// TIA Portal V18 export
FUNCTION_BLOCK "ST10_StopperCtrl"   // FB2601, LAD
TITLE = 输送带控制
{ S7_Optimized_Access := 'FALSE' }
VERSION : 0.1
// stored: AutoNumber false, IsIECCheckEnabled false, SetENOAutomatically false, UDAEnableTagReadback false
   VAR
      Stopper { S7_SetPoint := 'True'} : Array[1..100] of "StopperCtrl";
   END_VAR
   VAR_TEMP   // added for the SCL form of the ladder/FBD networks
      _w1 : Bool;
   END_VAR
BEGIN

REGION Network 1: ------------------------------------------------------------------------------------------------------------------------------ / ------------------------------------------------ H -------------------------------------------------------------------------
END_REGION

REGION Network 2: H-shaftLoadingStopperCylinder1
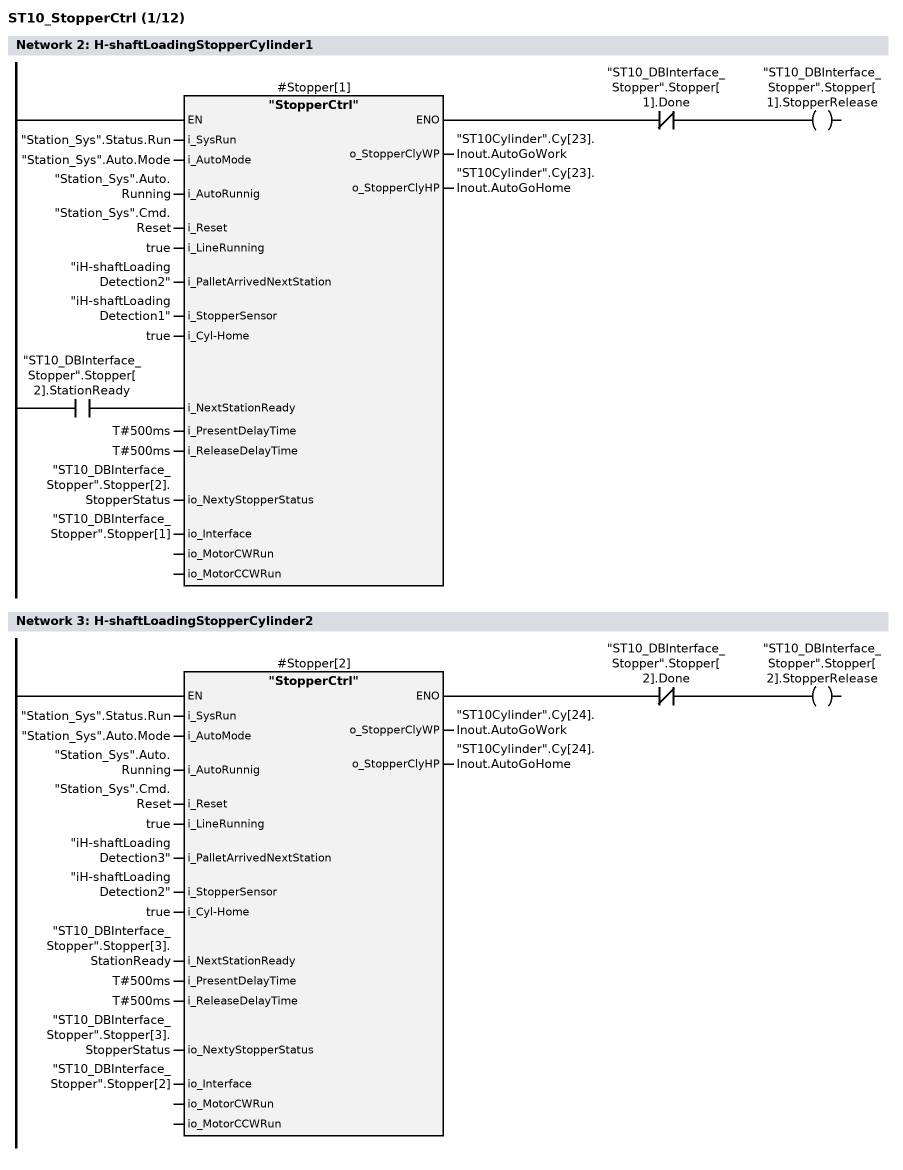
   RUNG wire#powerrail
      #Stopper[1](i_NextStationReady := wire#w1, i_SysRun := "Station_Sys".Status.Run, i_AutoMode := "Station_Sys".Auto.Mode, i_AutoRunnig := "Station_Sys".Auto.Running, i_Reset := "Station_Sys".Cmd.Reset, i_LineRunning := true, i_PalletArrivedNextStation := "iH-shaftLoadingDetection2", i_StopperSensor := "iH-shaftLoadingDetection1", "i_Cyl-Home" := true, i_PresentDelayTime := T#500ms, i_ReleaseDelayTime := T#500ms, io_NextyStopperStatus := "ST10_DBInterface_Stopper".Stopper[2].StopperStatus, io_Interface := "ST10_DBInterface_Stopper".Stopper[1], io_MotorCWRun :=, io_MotorCCWRun :=, o_StopperClyWP => "ST10Cylinder".Cy[23].Inout.AutoGoWork, o_StopperClyHP => "ST10Cylinder".Cy[23].Inout.AutoGoHome)
      I_Contact( "ST10_DBInterface_Stopper".Stopper[1].Done )
      Coil( "ST10_DBInterface_Stopper".Stopper[1].StopperRelease )
   END_RUNG
   RUNG wire#powerrail
      Contact( "ST10_DBInterface_Stopper".Stopper[2].StationReady )
   END_RUNG wire#w1
   // the same network as SCL:
   #Stopper[1](i_SysRun := "Station_Sys".Status.Run,   // "StopperCtrl"
               i_AutoMode := "Station_Sys".Auto.Mode,
               i_AutoRunnig := "Station_Sys".Auto.Running,
               i_Reset := "Station_Sys".Cmd.Reset,
               i_LineRunning := true,
               i_PalletArrivedNextStation := "iH-shaftLoadingDetection2",
               i_StopperSensor := "iH-shaftLoadingDetection1",
               "i_Cyl-Home" := true,
               i_NextStationReady := "ST10_DBInterface_Stopper".Stopper[2].StationReady,
               i_PresentDelayTime := T#500ms,
               i_ReleaseDelayTime := T#500ms,
               io_NextyStopperStatus := "ST10_DBInterface_Stopper".Stopper[2].StopperStatus,
               io_Interface := "ST10_DBInterface_Stopper".Stopper[1],
               o_StopperClyWP => "ST10Cylinder".Cy[23].Inout.AutoGoWork,
               o_StopperClyHP => "ST10Cylinder".Cy[23].Inout.AutoGoHome,
               ENO => #_w1);
   "ST10_DBInterface_Stopper".Stopper[1].StopperRelease := #_w1 AND NOT "ST10_DBInterface_Stopper".Stopper[1].Done;
END_REGION

REGION Network 3: H-shaftLoadingStopperCylinder2
   RUNG wire#powerrail
      #Stopper[2](i_SysRun := "Station_Sys".Status.Run, i_AutoMode := "Station_Sys".Auto.Mode, i_AutoRunnig := "Station_Sys".Auto.Running, i_Reset := "Station_Sys".Cmd.Reset, i_LineRunning := true, i_PalletArrivedNextStation := "iH-shaftLoadingDetection3", i_StopperSensor := "iH-shaftLoadingDetection2", "i_Cyl-Home" := true, i_NextStationReady := "ST10_DBInterface_Stopper".Stopper[3].StationReady, i_PresentDelayTime := T#500ms, i_ReleaseDelayTime := T#500ms, io_NextyStopperStatus := "ST10_DBInterface_Stopper".Stopper[3].StopperStatus, io_Interface := "ST10_DBInterface_Stopper".Stopper[2], io_MotorCWRun :=, io_MotorCCWRun :=, o_StopperClyWP => "ST10Cylinder".Cy[24].Inout.AutoGoWork, o_StopperClyHP => "ST10Cylinder".Cy[24].Inout.AutoGoHome)
      I_Contact( "ST10_DBInterface_Stopper".Stopper[2].Done )
      Coil( "ST10_DBInterface_Stopper".Stopper[2].StopperRelease )
   END_RUNG
   // the same network as SCL:
   #Stopper[2](i_SysRun := "Station_Sys".Status.Run,   // "StopperCtrl"
               i_AutoMode := "Station_Sys".Auto.Mode,
               i_AutoRunnig := "Station_Sys".Auto.Running,
               i_Reset := "Station_Sys".Cmd.Reset,
               i_LineRunning := true,
               i_PalletArrivedNextStation := "iH-shaftLoadingDetection3",
               i_StopperSensor := "iH-shaftLoadingDetection2",
               "i_Cyl-Home" := true,
               i_NextStationReady := "ST10_DBInterface_Stopper".Stopper[3].StationReady,
               i_PresentDelayTime := T#500ms,
               i_ReleaseDelayTime := T#500ms,
               io_NextyStopperStatus := "ST10_DBInterface_Stopper".Stopper[3].StopperStatus,
               io_Interface := "ST10_DBInterface_Stopper".Stopper[2],
               o_StopperClyWP => "ST10Cylinder".Cy[24].Inout.AutoGoWork,
               o_StopperClyHP => "ST10Cylinder".Cy[24].Inout.AutoGoHome,
               ENO => #_w1);
   "ST10_DBInterface_Stopper".Stopper[2].StopperRelease := #_w1 AND NOT "ST10_DBInterface_Stopper".Stopper[2].Done;
END_REGION

REGION Network 4: H-shaftLoadingStopperCylinder3
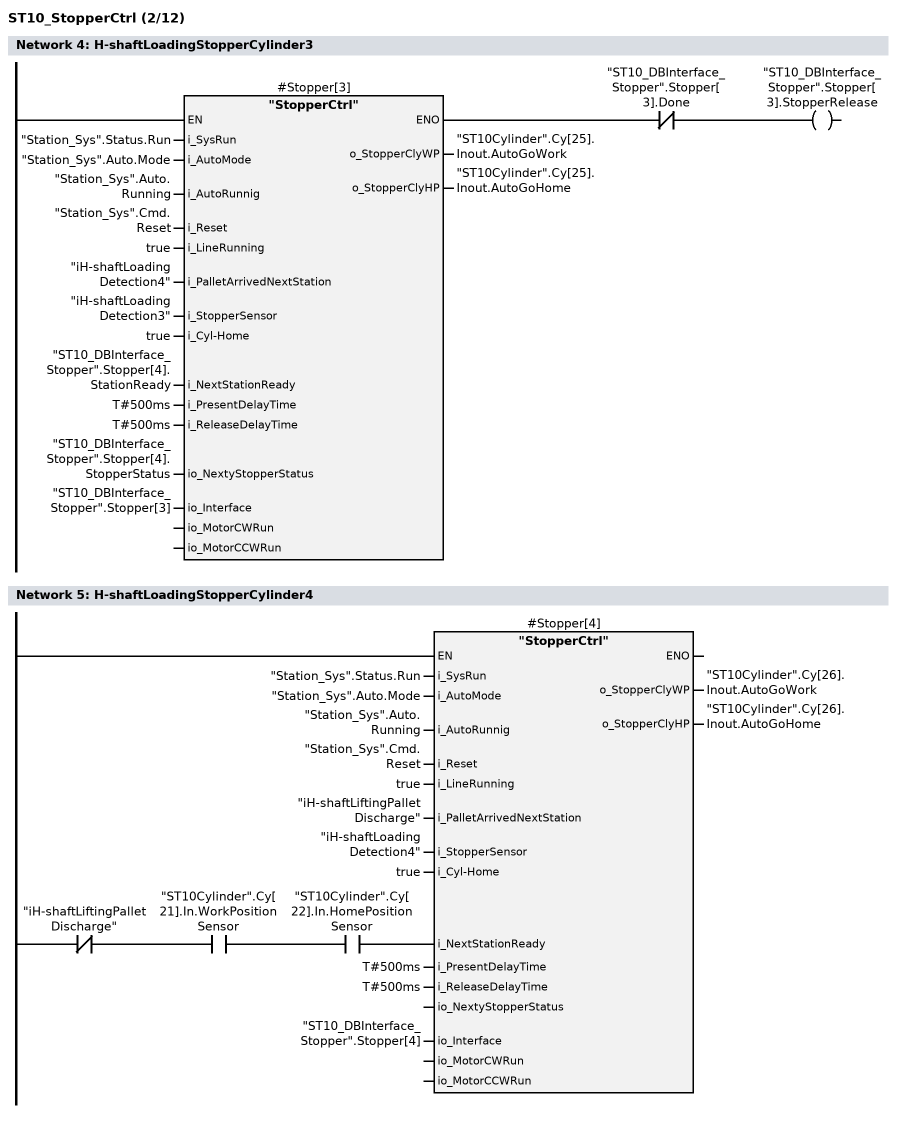
   RUNG wire#powerrail
      #Stopper[3](i_SysRun := "Station_Sys".Status.Run, i_AutoMode := "Station_Sys".Auto.Mode, i_AutoRunnig := "Station_Sys".Auto.Running, i_Reset := "Station_Sys".Cmd.Reset, i_LineRunning := true, i_PalletArrivedNextStation := "iH-shaftLoadingDetection4", i_StopperSensor := "iH-shaftLoadingDetection3", "i_Cyl-Home" := true, i_NextStationReady := "ST10_DBInterface_Stopper".Stopper[4].StationReady, i_PresentDelayTime := T#500ms, i_ReleaseDelayTime := T#500ms, io_NextyStopperStatus := "ST10_DBInterface_Stopper".Stopper[4].StopperStatus, io_Interface := "ST10_DBInterface_Stopper".Stopper[3], io_MotorCWRun :=, io_MotorCCWRun :=, o_StopperClyWP => "ST10Cylinder".Cy[25].Inout.AutoGoWork, o_StopperClyHP => "ST10Cylinder".Cy[25].Inout.AutoGoHome)
      I_Contact( "ST10_DBInterface_Stopper".Stopper[3].Done )
      Coil( "ST10_DBInterface_Stopper".Stopper[3].StopperRelease )
   END_RUNG
   // the same network as SCL:
   #Stopper[3](i_SysRun := "Station_Sys".Status.Run,   // "StopperCtrl"
               i_AutoMode := "Station_Sys".Auto.Mode,
               i_AutoRunnig := "Station_Sys".Auto.Running,
               i_Reset := "Station_Sys".Cmd.Reset,
               i_LineRunning := true,
               i_PalletArrivedNextStation := "iH-shaftLoadingDetection4",
               i_StopperSensor := "iH-shaftLoadingDetection3",
               "i_Cyl-Home" := true,
               i_NextStationReady := "ST10_DBInterface_Stopper".Stopper[4].StationReady,
               i_PresentDelayTime := T#500ms,
               i_ReleaseDelayTime := T#500ms,
               io_NextyStopperStatus := "ST10_DBInterface_Stopper".Stopper[4].StopperStatus,
               io_Interface := "ST10_DBInterface_Stopper".Stopper[3],
               o_StopperClyWP => "ST10Cylinder".Cy[25].Inout.AutoGoWork,
               o_StopperClyHP => "ST10Cylinder".Cy[25].Inout.AutoGoHome,
               ENO => #_w1);
   "ST10_DBInterface_Stopper".Stopper[3].StopperRelease := #_w1 AND NOT "ST10_DBInterface_Stopper".Stopper[3].Done;
END_REGION

REGION Network 5: H-shaftLoadingStopperCylinder4
   RUNG wire#powerrail
      #Stopper[4](i_NextStationReady := wire#w1, i_SysRun := "Station_Sys".Status.Run, i_AutoMode := "Station_Sys".Auto.Mode, i_AutoRunnig := "Station_Sys".Auto.Running, i_Reset := "Station_Sys".Cmd.Reset, i_LineRunning := true, i_PalletArrivedNextStation := "iH-shaftLiftingPalletDischarge", i_StopperSensor := "iH-shaftLoadingDetection4", "i_Cyl-Home" := true, i_PresentDelayTime := T#500ms, i_ReleaseDelayTime := T#500ms, io_NextyStopperStatus :=, io_Interface := "ST10_DBInterface_Stopper".Stopper[4], io_MotorCWRun :=, io_MotorCCWRun :=, o_StopperClyWP => "ST10Cylinder".Cy[26].Inout.AutoGoWork, o_StopperClyHP => "ST10Cylinder".Cy[26].Inout.AutoGoHome)
   END_RUNG
   RUNG wire#powerrail
      I_Contact( "iH-shaftLiftingPalletDischarge" )
      Contact( "ST10Cylinder".Cy[21].In.WorkPositionSensor )
      Contact( "ST10Cylinder".Cy[22].In.HomePositionSensor )
   END_RUNG wire#w1
   // the same network as SCL:
   #Stopper[4](i_SysRun := "Station_Sys".Status.Run,   // "StopperCtrl"
               i_AutoMode := "Station_Sys".Auto.Mode,
               i_AutoRunnig := "Station_Sys".Auto.Running,
               i_Reset := "Station_Sys".Cmd.Reset,
               i_LineRunning := true,
               i_PalletArrivedNextStation := "iH-shaftLiftingPalletDischarge",
               i_StopperSensor := "iH-shaftLoadingDetection4",
               "i_Cyl-Home" := true,
               i_NextStationReady := NOT "iH-shaftLiftingPalletDischarge" AND "ST10Cylinder".Cy[21].In.WorkPositionSensor AND "ST10Cylinder".Cy[22].In.HomePositionSensor,
               i_PresentDelayTime := T#500ms,
               i_ReleaseDelayTime := T#500ms,
               io_Interface := "ST10_DBInterface_Stopper".Stopper[4],
               o_StopperClyWP => "ST10Cylinder".Cy[26].Inout.AutoGoWork,
               o_StopperClyHP => "ST10Cylinder".Cy[26].Inout.AutoGoHome);
END_REGION

REGION Network 6: H-shaftTakeStopperCylinder1
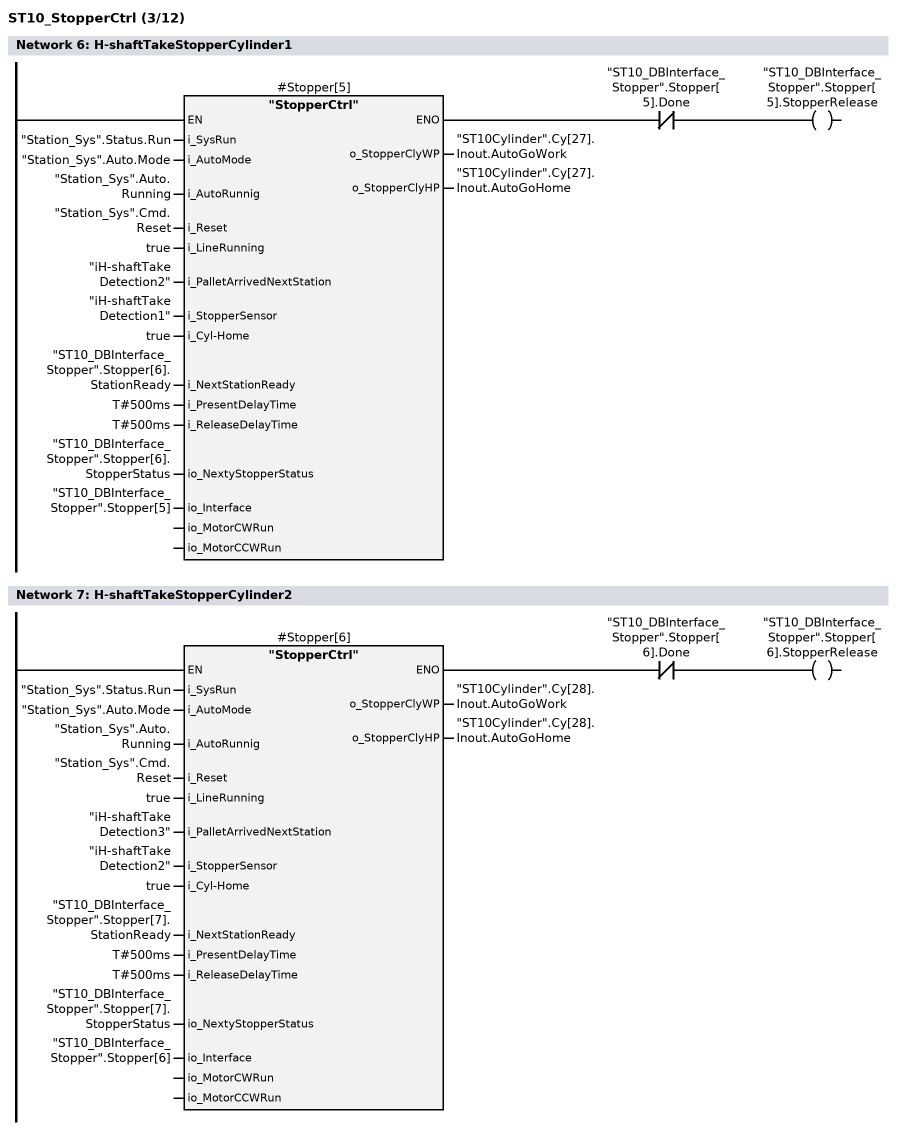
   RUNG wire#powerrail
      #Stopper[5](i_SysRun := "Station_Sys".Status.Run, i_AutoMode := "Station_Sys".Auto.Mode, i_AutoRunnig := "Station_Sys".Auto.Running, i_Reset := "Station_Sys".Cmd.Reset, i_LineRunning := true, i_PalletArrivedNextStation := "iH-shaftTakeDetection2", i_StopperSensor := "iH-shaftTakeDetection1", "i_Cyl-Home" := true, i_NextStationReady := "ST10_DBInterface_Stopper".Stopper[6].StationReady, i_PresentDelayTime := T#500ms, i_ReleaseDelayTime := T#500ms, io_NextyStopperStatus := "ST10_DBInterface_Stopper".Stopper[6].StopperStatus, io_Interface := "ST10_DBInterface_Stopper".Stopper[5], io_MotorCWRun :=, io_MotorCCWRun :=, o_StopperClyWP => "ST10Cylinder".Cy[27].Inout.AutoGoWork, o_StopperClyHP => "ST10Cylinder".Cy[27].Inout.AutoGoHome)
      I_Contact( "ST10_DBInterface_Stopper".Stopper[5].Done )
      Coil( "ST10_DBInterface_Stopper".Stopper[5].StopperRelease )
   END_RUNG
   // the same network as SCL:
   #Stopper[5](i_SysRun := "Station_Sys".Status.Run,   // "StopperCtrl"
               i_AutoMode := "Station_Sys".Auto.Mode,
               i_AutoRunnig := "Station_Sys".Auto.Running,
               i_Reset := "Station_Sys".Cmd.Reset,
               i_LineRunning := true,
               i_PalletArrivedNextStation := "iH-shaftTakeDetection2",
               i_StopperSensor := "iH-shaftTakeDetection1",
               "i_Cyl-Home" := true,
               i_NextStationReady := "ST10_DBInterface_Stopper".Stopper[6].StationReady,
               i_PresentDelayTime := T#500ms,
               i_ReleaseDelayTime := T#500ms,
               io_NextyStopperStatus := "ST10_DBInterface_Stopper".Stopper[6].StopperStatus,
               io_Interface := "ST10_DBInterface_Stopper".Stopper[5],
               o_StopperClyWP => "ST10Cylinder".Cy[27].Inout.AutoGoWork,
               o_StopperClyHP => "ST10Cylinder".Cy[27].Inout.AutoGoHome,
               ENO => #_w1);
   "ST10_DBInterface_Stopper".Stopper[5].StopperRelease := #_w1 AND NOT "ST10_DBInterface_Stopper".Stopper[5].Done;
END_REGION

REGION Network 7: H-shaftTakeStopperCylinder2
   RUNG wire#powerrail
      #Stopper[6](i_SysRun := "Station_Sys".Status.Run, i_AutoMode := "Station_Sys".Auto.Mode, i_AutoRunnig := "Station_Sys".Auto.Running, i_Reset := "Station_Sys".Cmd.Reset, i_LineRunning := true, i_PalletArrivedNextStation := "iH-shaftTakeDetection3", i_StopperSensor := "iH-shaftTakeDetection2", "i_Cyl-Home" := true, i_NextStationReady := "ST10_DBInterface_Stopper".Stopper[7].StationReady, i_PresentDelayTime := T#500ms, i_ReleaseDelayTime := T#500ms, io_NextyStopperStatus := "ST10_DBInterface_Stopper".Stopper[7].StopperStatus, io_Interface := "ST10_DBInterface_Stopper".Stopper[6], io_MotorCWRun :=, io_MotorCCWRun :=, o_StopperClyWP => "ST10Cylinder".Cy[28].Inout.AutoGoWork, o_StopperClyHP => "ST10Cylinder".Cy[28].Inout.AutoGoHome)
      I_Contact( "ST10_DBInterface_Stopper".Stopper[6].Done )
      Coil( "ST10_DBInterface_Stopper".Stopper[6].StopperRelease )
   END_RUNG
   // the same network as SCL:
   #Stopper[6](i_SysRun := "Station_Sys".Status.Run,   // "StopperCtrl"
               i_AutoMode := "Station_Sys".Auto.Mode,
               i_AutoRunnig := "Station_Sys".Auto.Running,
               i_Reset := "Station_Sys".Cmd.Reset,
               i_LineRunning := true,
               i_PalletArrivedNextStation := "iH-shaftTakeDetection3",
               i_StopperSensor := "iH-shaftTakeDetection2",
               "i_Cyl-Home" := true,
               i_NextStationReady := "ST10_DBInterface_Stopper".Stopper[7].StationReady,
               i_PresentDelayTime := T#500ms,
               i_ReleaseDelayTime := T#500ms,
               io_NextyStopperStatus := "ST10_DBInterface_Stopper".Stopper[7].StopperStatus,
               io_Interface := "ST10_DBInterface_Stopper".Stopper[6],
               o_StopperClyWP => "ST10Cylinder".Cy[28].Inout.AutoGoWork,
               o_StopperClyHP => "ST10Cylinder".Cy[28].Inout.AutoGoHome,
               ENO => #_w1);
   "ST10_DBInterface_Stopper".Stopper[6].StopperRelease := #_w1 AND NOT "ST10_DBInterface_Stopper".Stopper[6].Done;
END_REGION

REGION Network 8: H-shaftTakeStopperCylinder3
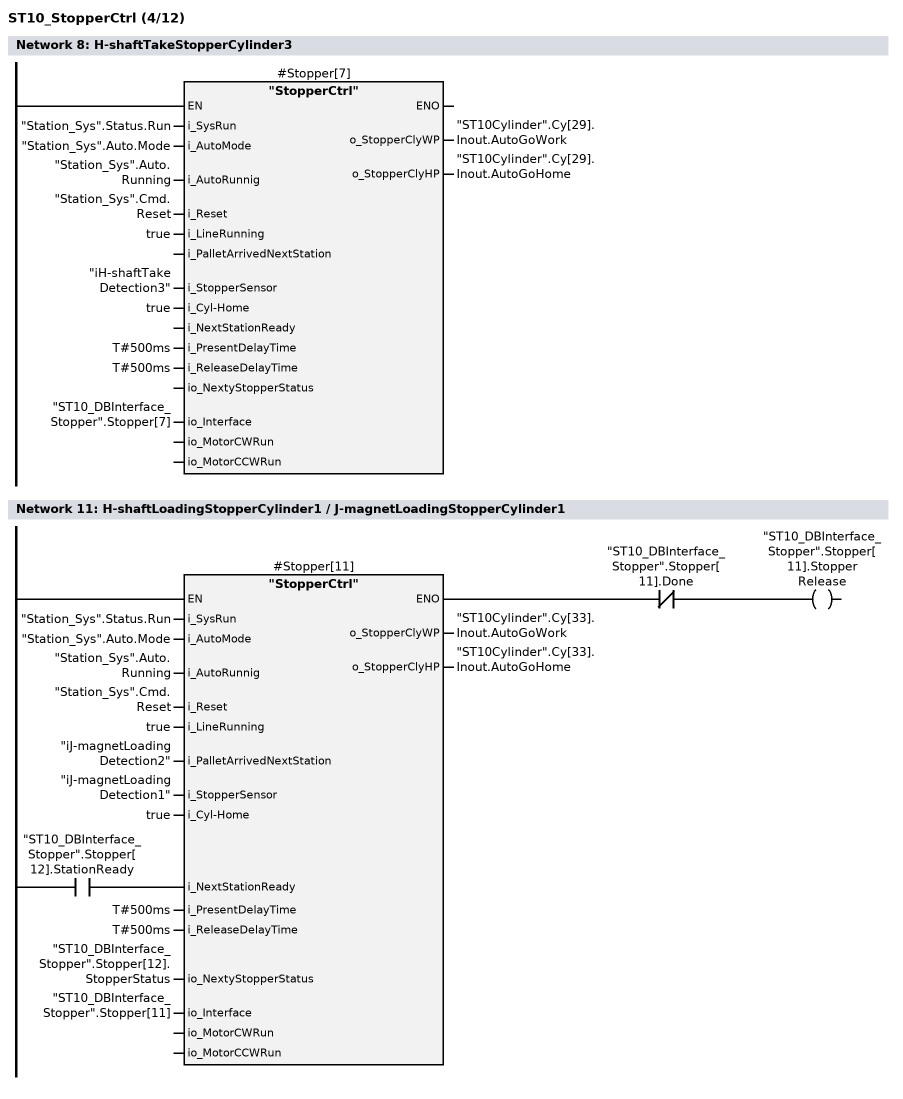
   RUNG wire#powerrail
      #Stopper[7](i_SysRun := "Station_Sys".Status.Run, i_AutoMode := "Station_Sys".Auto.Mode, i_AutoRunnig := "Station_Sys".Auto.Running, i_Reset := "Station_Sys".Cmd.Reset, i_LineRunning := true, i_PalletArrivedNextStation :=, i_StopperSensor := "iH-shaftTakeDetection3", "i_Cyl-Home" := true, i_NextStationReady :=, i_PresentDelayTime := T#500ms, i_ReleaseDelayTime := T#500ms, io_NextyStopperStatus :=, io_Interface := "ST10_DBInterface_Stopper".Stopper[7], io_MotorCWRun :=, io_MotorCCWRun :=, o_StopperClyWP => "ST10Cylinder".Cy[29].Inout.AutoGoWork, o_StopperClyHP => "ST10Cylinder".Cy[29].Inout.AutoGoHome)
   END_RUNG
   // the same network as SCL:
   #Stopper[7](i_SysRun := "Station_Sys".Status.Run,   // "StopperCtrl"
               i_AutoMode := "Station_Sys".Auto.Mode,
               i_AutoRunnig := "Station_Sys".Auto.Running,
               i_Reset := "Station_Sys".Cmd.Reset,
               i_LineRunning := true,
               i_StopperSensor := "iH-shaftTakeDetection3",
               "i_Cyl-Home" := true,
               i_PresentDelayTime := T#500ms,
               i_ReleaseDelayTime := T#500ms,
               io_Interface := "ST10_DBInterface_Stopper".Stopper[7],
               o_StopperClyWP => "ST10Cylinder".Cy[29].Inout.AutoGoWork,
               o_StopperClyHP => "ST10Cylinder".Cy[29].Inout.AutoGoHome);
END_REGION

REGION Network 9: -------------------------------------------------------------------------------------------------------------------------------
END_REGION

REGION Network 10: ------------------------------------------------------------------------------------------------------------------------------ / ------------------------------------------------ J -------------------------------------------------------------------------
END_REGION

REGION Network 11: H-shaftLoadingStopperCylinder1 / J-magnetLoadingStopperCylinder1
   RUNG wire#powerrail
      #Stopper[11](i_NextStationReady := wire#w1, i_SysRun := "Station_Sys".Status.Run, i_AutoMode := "Station_Sys".Auto.Mode, i_AutoRunnig := "Station_Sys".Auto.Running, i_Reset := "Station_Sys".Cmd.Reset, i_LineRunning := true, i_PalletArrivedNextStation := "iJ-magnetLoadingDetection2", i_StopperSensor := "iJ-magnetLoadingDetection1", "i_Cyl-Home" := true, i_PresentDelayTime := T#500ms, i_ReleaseDelayTime := T#500ms, io_NextyStopperStatus := "ST10_DBInterface_Stopper".Stopper[12].StopperStatus, io_Interface := "ST10_DBInterface_Stopper".Stopper[11], io_MotorCWRun :=, io_MotorCCWRun :=, o_StopperClyWP => "ST10Cylinder".Cy[33].Inout.AutoGoWork, o_StopperClyHP => "ST10Cylinder".Cy[33].Inout.AutoGoHome)
      I_Contact( "ST10_DBInterface_Stopper".Stopper[11].Done )
      Coil( "ST10_DBInterface_Stopper".Stopper[11].StopperRelease )
   END_RUNG
   RUNG wire#powerrail
      Contact( "ST10_DBInterface_Stopper".Stopper[12].StationReady )
   END_RUNG wire#w1
   // the same network as SCL:
   #Stopper[11](i_SysRun := "Station_Sys".Status.Run,   // "StopperCtrl"
                i_AutoMode := "Station_Sys".Auto.Mode,
                i_AutoRunnig := "Station_Sys".Auto.Running,
                i_Reset := "Station_Sys".Cmd.Reset,
                i_LineRunning := true,
                i_PalletArrivedNextStation := "iJ-magnetLoadingDetection2",
                i_StopperSensor := "iJ-magnetLoadingDetection1",
                "i_Cyl-Home" := true,
                i_NextStationReady := "ST10_DBInterface_Stopper".Stopper[12].StationReady,
                i_PresentDelayTime := T#500ms,
                i_ReleaseDelayTime := T#500ms,
                io_NextyStopperStatus := "ST10_DBInterface_Stopper".Stopper[12].StopperStatus,
                io_Interface := "ST10_DBInterface_Stopper".Stopper[11],
                o_StopperClyWP => "ST10Cylinder".Cy[33].Inout.AutoGoWork,
                o_StopperClyHP => "ST10Cylinder".Cy[33].Inout.AutoGoHome,
                ENO => #_w1);
   "ST10_DBInterface_Stopper".Stopper[11].StopperRelease := #_w1 AND NOT "ST10_DBInterface_Stopper".Stopper[11].Done;
END_REGION

REGION Network 12: H-shaftLoadingStopperCylinder2 / J-magnetLoadingStopperCylinder2
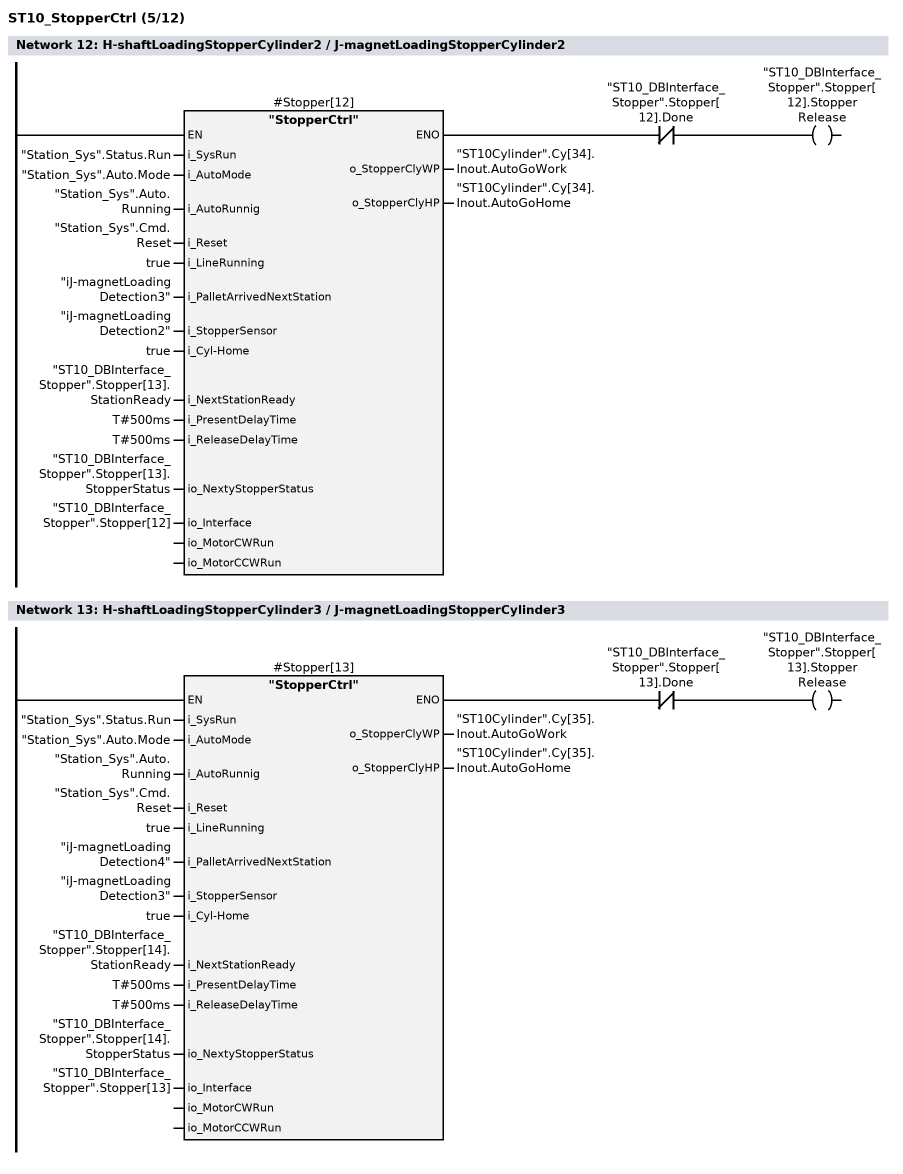
   RUNG wire#powerrail
      #Stopper[12](i_SysRun := "Station_Sys".Status.Run, i_AutoMode := "Station_Sys".Auto.Mode, i_AutoRunnig := "Station_Sys".Auto.Running, i_Reset := "Station_Sys".Cmd.Reset, i_LineRunning := true, i_PalletArrivedNextStation := "iJ-magnetLoadingDetection3", i_StopperSensor := "iJ-magnetLoadingDetection2", "i_Cyl-Home" := true, i_NextStationReady := "ST10_DBInterface_Stopper".Stopper[13].StationReady, i_PresentDelayTime := T#500ms, i_ReleaseDelayTime := T#500ms, io_NextyStopperStatus := "ST10_DBInterface_Stopper".Stopper[13].StopperStatus, io_Interface := "ST10_DBInterface_Stopper".Stopper[12], io_MotorCWRun :=, io_MotorCCWRun :=, o_StopperClyWP => "ST10Cylinder".Cy[34].Inout.AutoGoWork, o_StopperClyHP => "ST10Cylinder".Cy[34].Inout.AutoGoHome)
      I_Contact( "ST10_DBInterface_Stopper".Stopper[12].Done )
      Coil( "ST10_DBInterface_Stopper".Stopper[12].StopperRelease )
   END_RUNG
   // the same network as SCL:
   #Stopper[12](i_SysRun := "Station_Sys".Status.Run,   // "StopperCtrl"
                i_AutoMode := "Station_Sys".Auto.Mode,
                i_AutoRunnig := "Station_Sys".Auto.Running,
                i_Reset := "Station_Sys".Cmd.Reset,
                i_LineRunning := true,
                i_PalletArrivedNextStation := "iJ-magnetLoadingDetection3",
                i_StopperSensor := "iJ-magnetLoadingDetection2",
                "i_Cyl-Home" := true,
                i_NextStationReady := "ST10_DBInterface_Stopper".Stopper[13].StationReady,
                i_PresentDelayTime := T#500ms,
                i_ReleaseDelayTime := T#500ms,
                io_NextyStopperStatus := "ST10_DBInterface_Stopper".Stopper[13].StopperStatus,
                io_Interface := "ST10_DBInterface_Stopper".Stopper[12],
                o_StopperClyWP => "ST10Cylinder".Cy[34].Inout.AutoGoWork,
                o_StopperClyHP => "ST10Cylinder".Cy[34].Inout.AutoGoHome,
                ENO => #_w1);
   "ST10_DBInterface_Stopper".Stopper[12].StopperRelease := #_w1 AND NOT "ST10_DBInterface_Stopper".Stopper[12].Done;
END_REGION

REGION Network 13: H-shaftLoadingStopperCylinder3 / J-magnetLoadingStopperCylinder3
   RUNG wire#powerrail
      #Stopper[13](i_SysRun := "Station_Sys".Status.Run, i_AutoMode := "Station_Sys".Auto.Mode, i_AutoRunnig := "Station_Sys".Auto.Running, i_Reset := "Station_Sys".Cmd.Reset, i_LineRunning := true, i_PalletArrivedNextStation := "iJ-magnetLoadingDetection4", i_StopperSensor := "iJ-magnetLoadingDetection3", "i_Cyl-Home" := true, i_NextStationReady := "ST10_DBInterface_Stopper".Stopper[14].StationReady, i_PresentDelayTime := T#500ms, i_ReleaseDelayTime := T#500ms, io_NextyStopperStatus := "ST10_DBInterface_Stopper".Stopper[14].StopperStatus, io_Interface := "ST10_DBInterface_Stopper".Stopper[13], io_MotorCWRun :=, io_MotorCCWRun :=, o_StopperClyWP => "ST10Cylinder".Cy[35].Inout.AutoGoWork, o_StopperClyHP => "ST10Cylinder".Cy[35].Inout.AutoGoHome)
      I_Contact( "ST10_DBInterface_Stopper".Stopper[13].Done )
      Coil( "ST10_DBInterface_Stopper".Stopper[13].StopperRelease )
   END_RUNG
   // the same network as SCL:
   #Stopper[13](i_SysRun := "Station_Sys".Status.Run,   // "StopperCtrl"
                i_AutoMode := "Station_Sys".Auto.Mode,
                i_AutoRunnig := "Station_Sys".Auto.Running,
                i_Reset := "Station_Sys".Cmd.Reset,
                i_LineRunning := true,
                i_PalletArrivedNextStation := "iJ-magnetLoadingDetection4",
                i_StopperSensor := "iJ-magnetLoadingDetection3",
                "i_Cyl-Home" := true,
                i_NextStationReady := "ST10_DBInterface_Stopper".Stopper[14].StationReady,
                i_PresentDelayTime := T#500ms,
                i_ReleaseDelayTime := T#500ms,
                io_NextyStopperStatus := "ST10_DBInterface_Stopper".Stopper[14].StopperStatus,
                io_Interface := "ST10_DBInterface_Stopper".Stopper[13],
                o_StopperClyWP => "ST10Cylinder".Cy[35].Inout.AutoGoWork,
                o_StopperClyHP => "ST10Cylinder".Cy[35].Inout.AutoGoHome,
                ENO => #_w1);
   "ST10_DBInterface_Stopper".Stopper[13].StopperRelease := #_w1 AND NOT "ST10_DBInterface_Stopper".Stopper[13].Done;
END_REGION

REGION Network 14: H-shaftLoadingStopperCylinder4 / J-magnetLoadingStopperCylinder4
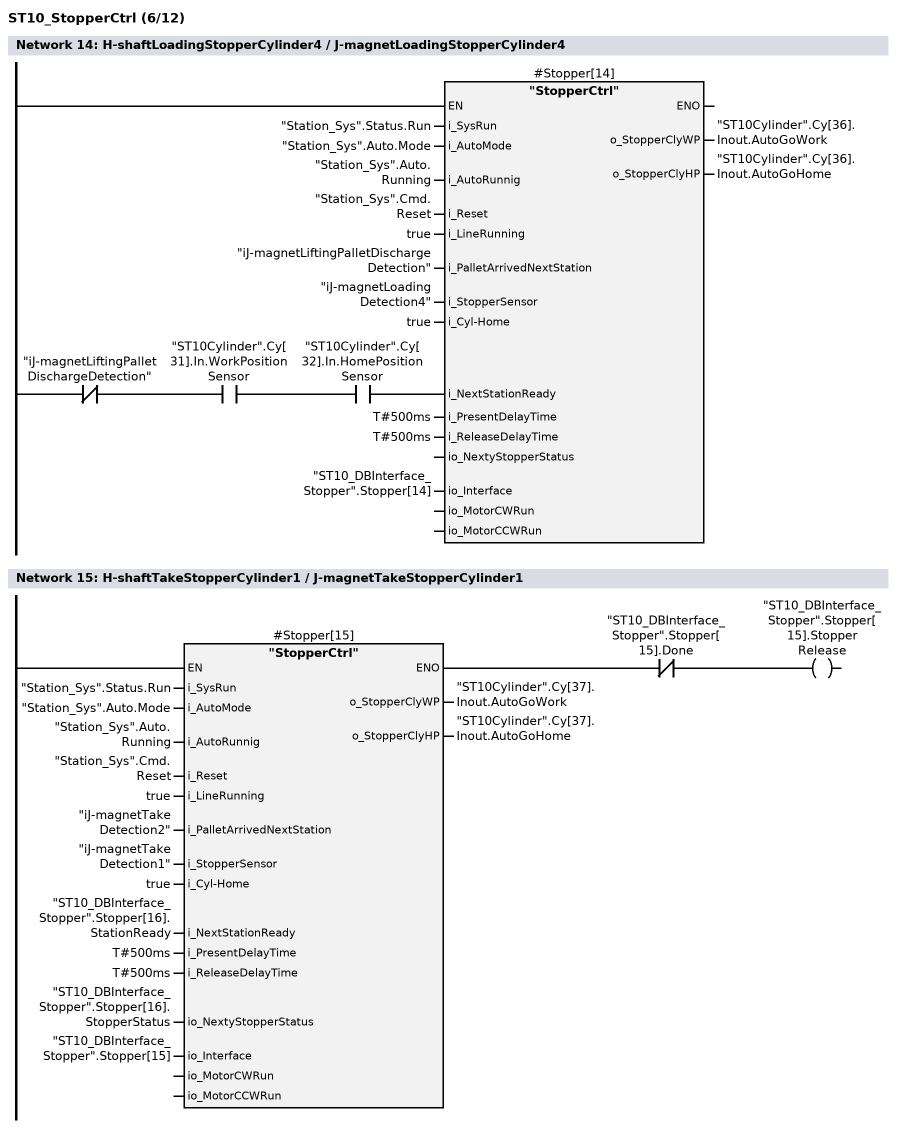
   RUNG wire#powerrail
      #Stopper[14](i_NextStationReady := wire#w1, i_SysRun := "Station_Sys".Status.Run, i_AutoMode := "Station_Sys".Auto.Mode, i_AutoRunnig := "Station_Sys".Auto.Running, i_Reset := "Station_Sys".Cmd.Reset, i_LineRunning := true, i_PalletArrivedNextStation := "iJ-magnetLiftingPalletDischargeDetection", i_StopperSensor := "iJ-magnetLoadingDetection4", "i_Cyl-Home" := true, i_PresentDelayTime := T#500ms, i_ReleaseDelayTime := T#500ms, io_NextyStopperStatus :=, io_Interface := "ST10_DBInterface_Stopper".Stopper[14], io_MotorCWRun :=, io_MotorCCWRun :=, o_StopperClyWP => "ST10Cylinder".Cy[36].Inout.AutoGoWork, o_StopperClyHP => "ST10Cylinder".Cy[36].Inout.AutoGoHome)
   END_RUNG
   RUNG wire#powerrail
      I_Contact( "iJ-magnetLiftingPalletDischargeDetection" )
      Contact( "ST10Cylinder".Cy[31].In.WorkPositionSensor )
      Contact( "ST10Cylinder".Cy[32].In.HomePositionSensor )
   END_RUNG wire#w1
   // the same network as SCL:
   #Stopper[14](i_SysRun := "Station_Sys".Status.Run,   // "StopperCtrl"
                i_AutoMode := "Station_Sys".Auto.Mode,
                i_AutoRunnig := "Station_Sys".Auto.Running,
                i_Reset := "Station_Sys".Cmd.Reset,
                i_LineRunning := true,
                i_PalletArrivedNextStation := "iJ-magnetLiftingPalletDischargeDetection",
                i_StopperSensor := "iJ-magnetLoadingDetection4",
                "i_Cyl-Home" := true,
                i_NextStationReady := NOT "iJ-magnetLiftingPalletDischargeDetection" AND "ST10Cylinder".Cy[31].In.WorkPositionSensor AND "ST10Cylinder".Cy[32].In.HomePositionSensor,
                i_PresentDelayTime := T#500ms,
                i_ReleaseDelayTime := T#500ms,
                io_Interface := "ST10_DBInterface_Stopper".Stopper[14],
                o_StopperClyWP => "ST10Cylinder".Cy[36].Inout.AutoGoWork,
                o_StopperClyHP => "ST10Cylinder".Cy[36].Inout.AutoGoHome);
END_REGION

REGION Network 15: H-shaftTakeStopperCylinder1 / J-magnetTakeStopperCylinder1
   RUNG wire#powerrail
      #Stopper[15](i_SysRun := "Station_Sys".Status.Run, i_AutoMode := "Station_Sys".Auto.Mode, i_AutoRunnig := "Station_Sys".Auto.Running, i_Reset := "Station_Sys".Cmd.Reset, i_LineRunning := true, i_PalletArrivedNextStation := "iJ-magnetTakeDetection2", i_StopperSensor := "iJ-magnetTakeDetection1", "i_Cyl-Home" := true, i_NextStationReady := "ST10_DBInterface_Stopper".Stopper[16].StationReady, i_PresentDelayTime := T#500ms, i_ReleaseDelayTime := T#500ms, io_NextyStopperStatus := "ST10_DBInterface_Stopper".Stopper[16].StopperStatus, io_Interface := "ST10_DBInterface_Stopper".Stopper[15], io_MotorCWRun :=, io_MotorCCWRun :=, o_StopperClyWP => "ST10Cylinder".Cy[37].Inout.AutoGoWork, o_StopperClyHP => "ST10Cylinder".Cy[37].Inout.AutoGoHome)
      I_Contact( "ST10_DBInterface_Stopper".Stopper[15].Done )
      Coil( "ST10_DBInterface_Stopper".Stopper[15].StopperRelease )
   END_RUNG
   // the same network as SCL:
   #Stopper[15](i_SysRun := "Station_Sys".Status.Run,   // "StopperCtrl"
                i_AutoMode := "Station_Sys".Auto.Mode,
                i_AutoRunnig := "Station_Sys".Auto.Running,
                i_Reset := "Station_Sys".Cmd.Reset,
                i_LineRunning := true,
                i_PalletArrivedNextStation := "iJ-magnetTakeDetection2",
                i_StopperSensor := "iJ-magnetTakeDetection1",
                "i_Cyl-Home" := true,
                i_NextStationReady := "ST10_DBInterface_Stopper".Stopper[16].StationReady,
                i_PresentDelayTime := T#500ms,
                i_ReleaseDelayTime := T#500ms,
                io_NextyStopperStatus := "ST10_DBInterface_Stopper".Stopper[16].StopperStatus,
                io_Interface := "ST10_DBInterface_Stopper".Stopper[15],
                o_StopperClyWP => "ST10Cylinder".Cy[37].Inout.AutoGoWork,
                o_StopperClyHP => "ST10Cylinder".Cy[37].Inout.AutoGoHome,
                ENO => #_w1);
   "ST10_DBInterface_Stopper".Stopper[15].StopperRelease := #_w1 AND NOT "ST10_DBInterface_Stopper".Stopper[15].Done;
END_REGION

REGION Network 16: H-shaftTakeStopperCylinder2 / J-magnetTakeStopperCylinder2
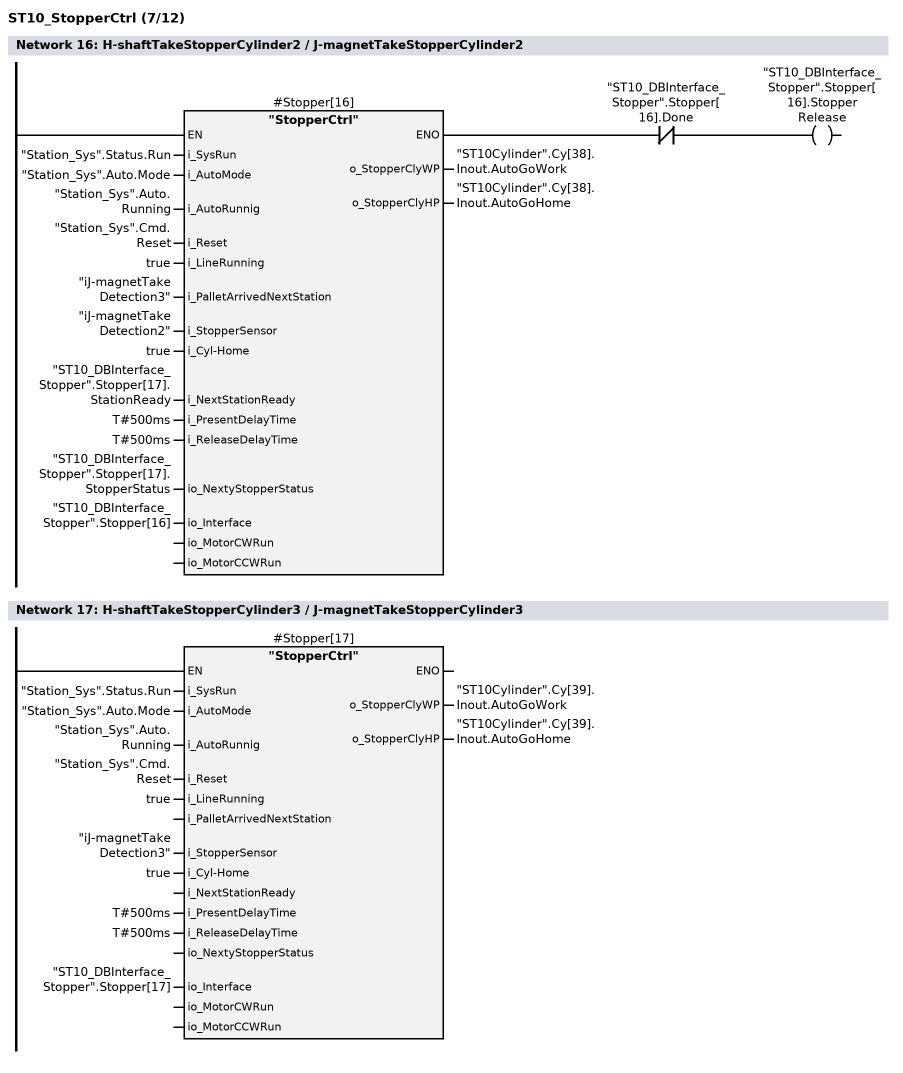
   RUNG wire#powerrail
      #Stopper[16](i_SysRun := "Station_Sys".Status.Run, i_AutoMode := "Station_Sys".Auto.Mode, i_AutoRunnig := "Station_Sys".Auto.Running, i_Reset := "Station_Sys".Cmd.Reset, i_LineRunning := true, i_PalletArrivedNextStation := "iJ-magnetTakeDetection3", i_StopperSensor := "iJ-magnetTakeDetection2", "i_Cyl-Home" := true, i_NextStationReady := "ST10_DBInterface_Stopper".Stopper[17].StationReady, i_PresentDelayTime := T#500ms, i_ReleaseDelayTime := T#500ms, io_NextyStopperStatus := "ST10_DBInterface_Stopper".Stopper[17].StopperStatus, io_Interface := "ST10_DBInterface_Stopper".Stopper[16], io_MotorCWRun :=, io_MotorCCWRun :=, o_StopperClyWP => "ST10Cylinder".Cy[38].Inout.AutoGoWork, o_StopperClyHP => "ST10Cylinder".Cy[38].Inout.AutoGoHome)
      I_Contact( "ST10_DBInterface_Stopper".Stopper[16].Done )
      Coil( "ST10_DBInterface_Stopper".Stopper[16].StopperRelease )
   END_RUNG
   // the same network as SCL:
   #Stopper[16](i_SysRun := "Station_Sys".Status.Run,   // "StopperCtrl"
                i_AutoMode := "Station_Sys".Auto.Mode,
                i_AutoRunnig := "Station_Sys".Auto.Running,
                i_Reset := "Station_Sys".Cmd.Reset,
                i_LineRunning := true,
                i_PalletArrivedNextStation := "iJ-magnetTakeDetection3",
                i_StopperSensor := "iJ-magnetTakeDetection2",
                "i_Cyl-Home" := true,
                i_NextStationReady := "ST10_DBInterface_Stopper".Stopper[17].StationReady,
                i_PresentDelayTime := T#500ms,
                i_ReleaseDelayTime := T#500ms,
                io_NextyStopperStatus := "ST10_DBInterface_Stopper".Stopper[17].StopperStatus,
                io_Interface := "ST10_DBInterface_Stopper".Stopper[16],
                o_StopperClyWP => "ST10Cylinder".Cy[38].Inout.AutoGoWork,
                o_StopperClyHP => "ST10Cylinder".Cy[38].Inout.AutoGoHome,
                ENO => #_w1);
   "ST10_DBInterface_Stopper".Stopper[16].StopperRelease := #_w1 AND NOT "ST10_DBInterface_Stopper".Stopper[16].Done;
END_REGION

REGION Network 17: H-shaftTakeStopperCylinder3 / J-magnetTakeStopperCylinder3
   RUNG wire#powerrail
      #Stopper[17](i_SysRun := "Station_Sys".Status.Run, i_AutoMode := "Station_Sys".Auto.Mode, i_AutoRunnig := "Station_Sys".Auto.Running, i_Reset := "Station_Sys".Cmd.Reset, i_LineRunning := true, i_PalletArrivedNextStation :=, i_StopperSensor := "iJ-magnetTakeDetection3", "i_Cyl-Home" := true, i_NextStationReady :=, i_PresentDelayTime := T#500ms, i_ReleaseDelayTime := T#500ms, io_NextyStopperStatus :=, io_Interface := "ST10_DBInterface_Stopper".Stopper[17], io_MotorCWRun :=, io_MotorCCWRun :=, o_StopperClyWP => "ST10Cylinder".Cy[39].Inout.AutoGoWork, o_StopperClyHP => "ST10Cylinder".Cy[39].Inout.AutoGoHome)
   END_RUNG
   // the same network as SCL:
   #Stopper[17](i_SysRun := "Station_Sys".Status.Run,   // "StopperCtrl"
                i_AutoMode := "Station_Sys".Auto.Mode,
                i_AutoRunnig := "Station_Sys".Auto.Running,
                i_Reset := "Station_Sys".Cmd.Reset,
                i_LineRunning := true,
                i_StopperSensor := "iJ-magnetTakeDetection3",
                "i_Cyl-Home" := true,
                i_PresentDelayTime := T#500ms,
                i_ReleaseDelayTime := T#500ms,
                io_Interface := "ST10_DBInterface_Stopper".Stopper[17],
                o_StopperClyWP => "ST10Cylinder".Cy[39].Inout.AutoGoWork,
                o_StopperClyHP => "ST10Cylinder".Cy[39].Inout.AutoGoHome);
END_REGION

REGION Network 18: -------------------------------------------------------------------------------------------------------------------------------
END_REGION

REGION Network 19: ------------------------------------------------------------------------------------------------------------------------------ / ------------------------------------------------ K -------------------------------------------------------------------------
END_REGION

REGION Network 20: H-shaftLoadingStopperCylinder1 / K-reserveLoadingStopperCylinder1
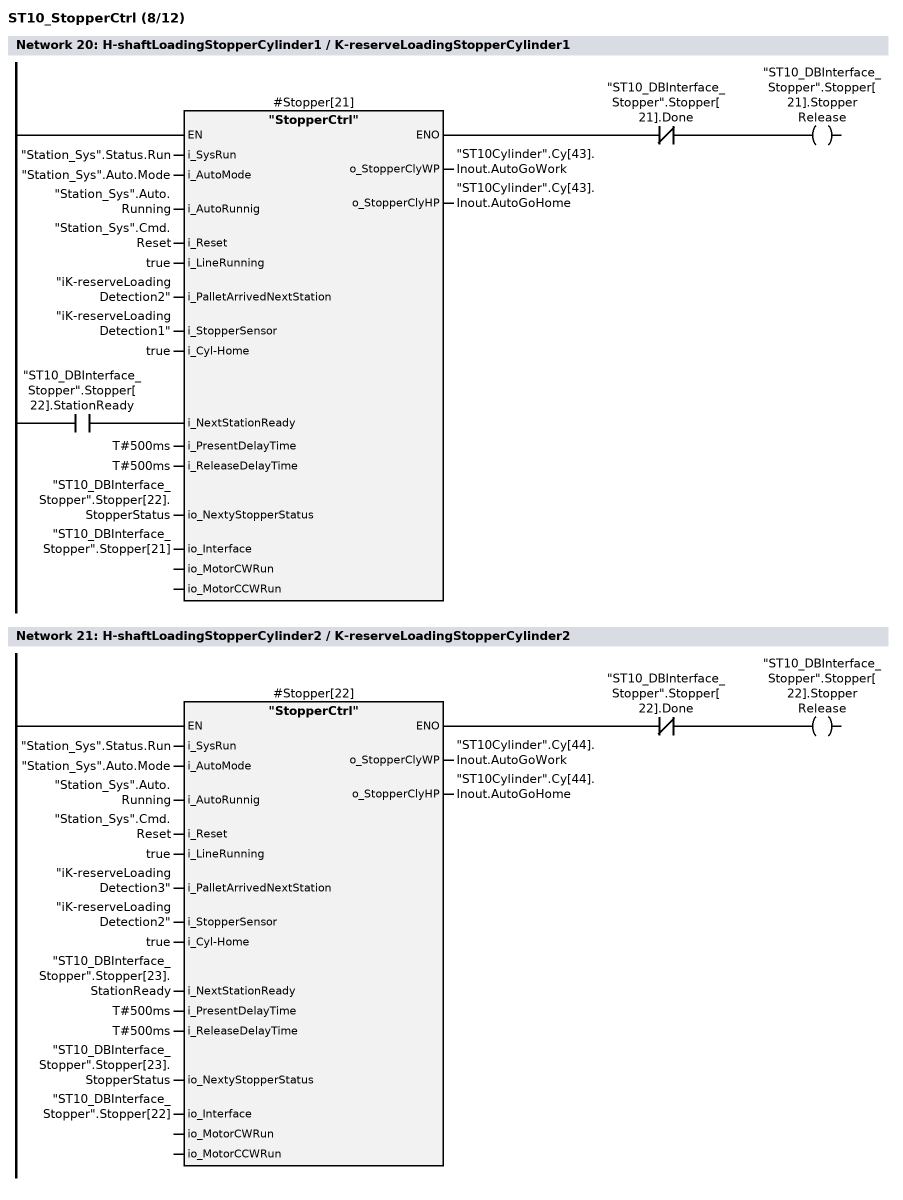
   RUNG wire#powerrail
      #Stopper[21](i_NextStationReady := wire#w1, i_SysRun := "Station_Sys".Status.Run, i_AutoMode := "Station_Sys".Auto.Mode, i_AutoRunnig := "Station_Sys".Auto.Running, i_Reset := "Station_Sys".Cmd.Reset, i_LineRunning := true, i_PalletArrivedNextStation := "iK-reserveLoadingDetection2", i_StopperSensor := "iK-reserveLoadingDetection1", "i_Cyl-Home" := true, i_PresentDelayTime := T#500ms, i_ReleaseDelayTime := T#500ms, io_NextyStopperStatus := "ST10_DBInterface_Stopper".Stopper[22].StopperStatus, io_Interface := "ST10_DBInterface_Stopper".Stopper[21], io_MotorCWRun :=, io_MotorCCWRun :=, o_StopperClyWP => "ST10Cylinder".Cy[43].Inout.AutoGoWork, o_StopperClyHP => "ST10Cylinder".Cy[43].Inout.AutoGoHome)
      I_Contact( "ST10_DBInterface_Stopper".Stopper[21].Done )
      Coil( "ST10_DBInterface_Stopper".Stopper[21].StopperRelease )
   END_RUNG
   RUNG wire#powerrail
      Contact( "ST10_DBInterface_Stopper".Stopper[22].StationReady )
   END_RUNG wire#w1
   // the same network as SCL:
   #Stopper[21](i_SysRun := "Station_Sys".Status.Run,   // "StopperCtrl"
                i_AutoMode := "Station_Sys".Auto.Mode,
                i_AutoRunnig := "Station_Sys".Auto.Running,
                i_Reset := "Station_Sys".Cmd.Reset,
                i_LineRunning := true,
                i_PalletArrivedNextStation := "iK-reserveLoadingDetection2",
                i_StopperSensor := "iK-reserveLoadingDetection1",
                "i_Cyl-Home" := true,
                i_NextStationReady := "ST10_DBInterface_Stopper".Stopper[22].StationReady,
                i_PresentDelayTime := T#500ms,
                i_ReleaseDelayTime := T#500ms,
                io_NextyStopperStatus := "ST10_DBInterface_Stopper".Stopper[22].StopperStatus,
                io_Interface := "ST10_DBInterface_Stopper".Stopper[21],
                o_StopperClyWP => "ST10Cylinder".Cy[43].Inout.AutoGoWork,
                o_StopperClyHP => "ST10Cylinder".Cy[43].Inout.AutoGoHome,
                ENO => #_w1);
   "ST10_DBInterface_Stopper".Stopper[21].StopperRelease := #_w1 AND NOT "ST10_DBInterface_Stopper".Stopper[21].Done;
END_REGION

REGION Network 21: H-shaftLoadingStopperCylinder2 / K-reserveLoadingStopperCylinder2
   RUNG wire#powerrail
      #Stopper[22](i_SysRun := "Station_Sys".Status.Run, i_AutoMode := "Station_Sys".Auto.Mode, i_AutoRunnig := "Station_Sys".Auto.Running, i_Reset := "Station_Sys".Cmd.Reset, i_LineRunning := true, i_PalletArrivedNextStation := "iK-reserveLoadingDetection3", i_StopperSensor := "iK-reserveLoadingDetection2", "i_Cyl-Home" := true, i_NextStationReady := "ST10_DBInterface_Stopper".Stopper[23].StationReady, i_PresentDelayTime := T#500ms, i_ReleaseDelayTime := T#500ms, io_NextyStopperStatus := "ST10_DBInterface_Stopper".Stopper[23].StopperStatus, io_Interface := "ST10_DBInterface_Stopper".Stopper[22], io_MotorCWRun :=, io_MotorCCWRun :=, o_StopperClyWP => "ST10Cylinder".Cy[44].Inout.AutoGoWork, o_StopperClyHP => "ST10Cylinder".Cy[44].Inout.AutoGoHome)
      I_Contact( "ST10_DBInterface_Stopper".Stopper[22].Done )
      Coil( "ST10_DBInterface_Stopper".Stopper[22].StopperRelease )
   END_RUNG
   // the same network as SCL:
   #Stopper[22](i_SysRun := "Station_Sys".Status.Run,   // "StopperCtrl"
                i_AutoMode := "Station_Sys".Auto.Mode,
                i_AutoRunnig := "Station_Sys".Auto.Running,
                i_Reset := "Station_Sys".Cmd.Reset,
                i_LineRunning := true,
                i_PalletArrivedNextStation := "iK-reserveLoadingDetection3",
                i_StopperSensor := "iK-reserveLoadingDetection2",
                "i_Cyl-Home" := true,
                i_NextStationReady := "ST10_DBInterface_Stopper".Stopper[23].StationReady,
                i_PresentDelayTime := T#500ms,
                i_ReleaseDelayTime := T#500ms,
                io_NextyStopperStatus := "ST10_DBInterface_Stopper".Stopper[23].StopperStatus,
                io_Interface := "ST10_DBInterface_Stopper".Stopper[22],
                o_StopperClyWP => "ST10Cylinder".Cy[44].Inout.AutoGoWork,
                o_StopperClyHP => "ST10Cylinder".Cy[44].Inout.AutoGoHome,
                ENO => #_w1);
   "ST10_DBInterface_Stopper".Stopper[22].StopperRelease := #_w1 AND NOT "ST10_DBInterface_Stopper".Stopper[22].Done;
END_REGION

REGION Network 22: H-shaftLoadingStopperCylinder3 / K-reserveLoadingStopperCylinder3
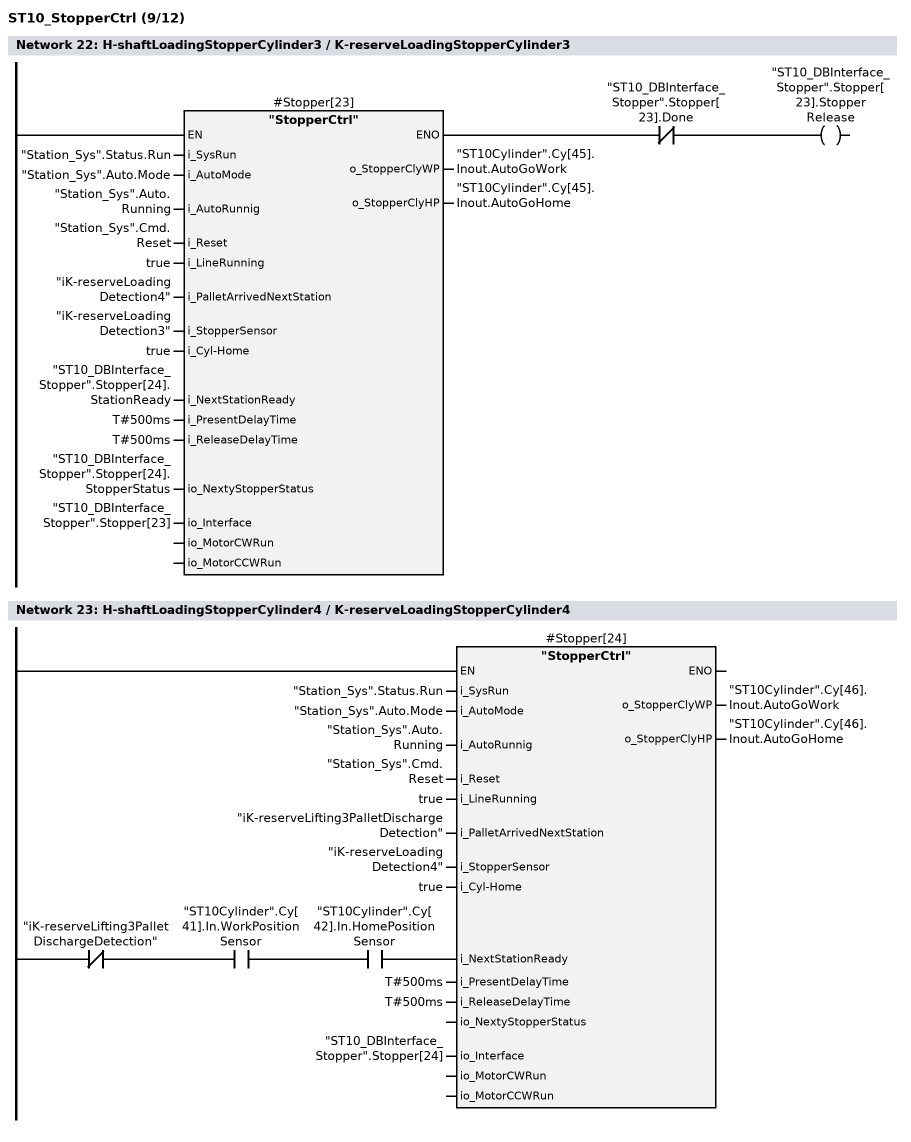
   RUNG wire#powerrail
      #Stopper[23](i_SysRun := "Station_Sys".Status.Run, i_AutoMode := "Station_Sys".Auto.Mode, i_AutoRunnig := "Station_Sys".Auto.Running, i_Reset := "Station_Sys".Cmd.Reset, i_LineRunning := true, i_PalletArrivedNextStation := "iK-reserveLoadingDetection4", i_StopperSensor := "iK-reserveLoadingDetection3", "i_Cyl-Home" := true, i_NextStationReady := "ST10_DBInterface_Stopper".Stopper[24].StationReady, i_PresentDelayTime := T#500ms, i_ReleaseDelayTime := T#500ms, io_NextyStopperStatus := "ST10_DBInterface_Stopper".Stopper[24].StopperStatus, io_Interface := "ST10_DBInterface_Stopper".Stopper[23], io_MotorCWRun :=, io_MotorCCWRun :=, o_StopperClyWP => "ST10Cylinder".Cy[45].Inout.AutoGoWork, o_StopperClyHP => "ST10Cylinder".Cy[45].Inout.AutoGoHome)
      I_Contact( "ST10_DBInterface_Stopper".Stopper[23].Done )
      Coil( "ST10_DBInterface_Stopper".Stopper[23].StopperRelease )
   END_RUNG
   // the same network as SCL:
   #Stopper[23](i_SysRun := "Station_Sys".Status.Run,   // "StopperCtrl"
                i_AutoMode := "Station_Sys".Auto.Mode,
                i_AutoRunnig := "Station_Sys".Auto.Running,
                i_Reset := "Station_Sys".Cmd.Reset,
                i_LineRunning := true,
                i_PalletArrivedNextStation := "iK-reserveLoadingDetection4",
                i_StopperSensor := "iK-reserveLoadingDetection3",
                "i_Cyl-Home" := true,
                i_NextStationReady := "ST10_DBInterface_Stopper".Stopper[24].StationReady,
                i_PresentDelayTime := T#500ms,
                i_ReleaseDelayTime := T#500ms,
                io_NextyStopperStatus := "ST10_DBInterface_Stopper".Stopper[24].StopperStatus,
                io_Interface := "ST10_DBInterface_Stopper".Stopper[23],
                o_StopperClyWP => "ST10Cylinder".Cy[45].Inout.AutoGoWork,
                o_StopperClyHP => "ST10Cylinder".Cy[45].Inout.AutoGoHome,
                ENO => #_w1);
   "ST10_DBInterface_Stopper".Stopper[23].StopperRelease := #_w1 AND NOT "ST10_DBInterface_Stopper".Stopper[23].Done;
END_REGION

REGION Network 23: H-shaftLoadingStopperCylinder4 / K-reserveLoadingStopperCylinder4
   RUNG wire#powerrail
      #Stopper[24](i_NextStationReady := wire#w1, i_SysRun := "Station_Sys".Status.Run, i_AutoMode := "Station_Sys".Auto.Mode, i_AutoRunnig := "Station_Sys".Auto.Running, i_Reset := "Station_Sys".Cmd.Reset, i_LineRunning := true, i_PalletArrivedNextStation := "iK-reserveLifting3PalletDischargeDetection", i_StopperSensor := "iK-reserveLoadingDetection4", "i_Cyl-Home" := true, i_PresentDelayTime := T#500ms, i_ReleaseDelayTime := T#500ms, io_NextyStopperStatus :=, io_Interface := "ST10_DBInterface_Stopper".Stopper[24], io_MotorCWRun :=, io_MotorCCWRun :=, o_StopperClyWP => "ST10Cylinder".Cy[46].Inout.AutoGoWork, o_StopperClyHP => "ST10Cylinder".Cy[46].Inout.AutoGoHome)
   END_RUNG
   RUNG wire#powerrail
      I_Contact( "iK-reserveLifting3PalletDischargeDetection" )
      Contact( "ST10Cylinder".Cy[41].In.WorkPositionSensor )
      Contact( "ST10Cylinder".Cy[42].In.HomePositionSensor )
   END_RUNG wire#w1
   // the same network as SCL:
   #Stopper[24](i_SysRun := "Station_Sys".Status.Run,   // "StopperCtrl"
                i_AutoMode := "Station_Sys".Auto.Mode,
                i_AutoRunnig := "Station_Sys".Auto.Running,
                i_Reset := "Station_Sys".Cmd.Reset,
                i_LineRunning := true,
                i_PalletArrivedNextStation := "iK-reserveLifting3PalletDischargeDetection",
                i_StopperSensor := "iK-reserveLoadingDetection4",
                "i_Cyl-Home" := true,
                i_NextStationReady := NOT "iK-reserveLifting3PalletDischargeDetection" AND "ST10Cylinder".Cy[41].In.WorkPositionSensor AND "ST10Cylinder".Cy[42].In.HomePositionSensor,
                i_PresentDelayTime := T#500ms,
                i_ReleaseDelayTime := T#500ms,
                io_Interface := "ST10_DBInterface_Stopper".Stopper[24],
                o_StopperClyWP => "ST10Cylinder".Cy[46].Inout.AutoGoWork,
                o_StopperClyHP => "ST10Cylinder".Cy[46].Inout.AutoGoHome);
END_REGION

REGION Network 24: H-shaftTakeStopperCylinder1 / K-reserveTakeStopperCylinder1
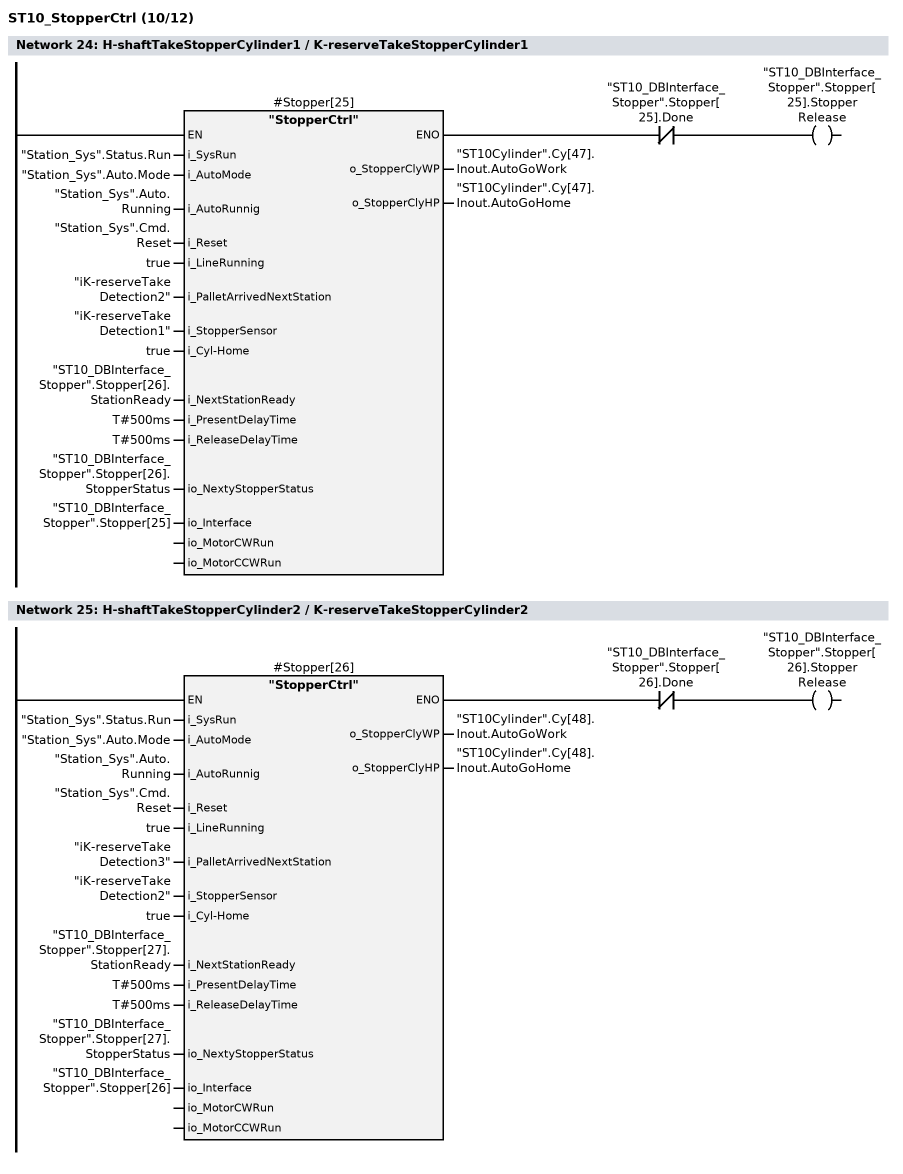
   RUNG wire#powerrail
      #Stopper[25](i_SysRun := "Station_Sys".Status.Run, i_AutoMode := "Station_Sys".Auto.Mode, i_AutoRunnig := "Station_Sys".Auto.Running, i_Reset := "Station_Sys".Cmd.Reset, i_LineRunning := true, i_PalletArrivedNextStation := "iK-reserveTakeDetection2", i_StopperSensor := "iK-reserveTakeDetection1", "i_Cyl-Home" := true, i_NextStationReady := "ST10_DBInterface_Stopper".Stopper[26].StationReady, i_PresentDelayTime := T#500ms, i_ReleaseDelayTime := T#500ms, io_NextyStopperStatus := "ST10_DBInterface_Stopper".Stopper[26].StopperStatus, io_Interface := "ST10_DBInterface_Stopper".Stopper[25], io_MotorCWRun :=, io_MotorCCWRun :=, o_StopperClyWP => "ST10Cylinder".Cy[47].Inout.AutoGoWork, o_StopperClyHP => "ST10Cylinder".Cy[47].Inout.AutoGoHome)
      I_Contact( "ST10_DBInterface_Stopper".Stopper[25].Done )
      Coil( "ST10_DBInterface_Stopper".Stopper[25].StopperRelease )
   END_RUNG
   // the same network as SCL:
   #Stopper[25](i_SysRun := "Station_Sys".Status.Run,   // "StopperCtrl"
                i_AutoMode := "Station_Sys".Auto.Mode,
                i_AutoRunnig := "Station_Sys".Auto.Running,
                i_Reset := "Station_Sys".Cmd.Reset,
                i_LineRunning := true,
                i_PalletArrivedNextStation := "iK-reserveTakeDetection2",
                i_StopperSensor := "iK-reserveTakeDetection1",
                "i_Cyl-Home" := true,
                i_NextStationReady := "ST10_DBInterface_Stopper".Stopper[26].StationReady,
                i_PresentDelayTime := T#500ms,
                i_ReleaseDelayTime := T#500ms,
                io_NextyStopperStatus := "ST10_DBInterface_Stopper".Stopper[26].StopperStatus,
                io_Interface := "ST10_DBInterface_Stopper".Stopper[25],
                o_StopperClyWP => "ST10Cylinder".Cy[47].Inout.AutoGoWork,
                o_StopperClyHP => "ST10Cylinder".Cy[47].Inout.AutoGoHome,
                ENO => #_w1);
   "ST10_DBInterface_Stopper".Stopper[25].StopperRelease := #_w1 AND NOT "ST10_DBInterface_Stopper".Stopper[25].Done;
END_REGION

REGION Network 25: H-shaftTakeStopperCylinder2 / K-reserveTakeStopperCylinder2
   RUNG wire#powerrail
      #Stopper[26](i_SysRun := "Station_Sys".Status.Run, i_AutoMode := "Station_Sys".Auto.Mode, i_AutoRunnig := "Station_Sys".Auto.Running, i_Reset := "Station_Sys".Cmd.Reset, i_LineRunning := true, i_PalletArrivedNextStation := "iK-reserveTakeDetection3", i_StopperSensor := "iK-reserveTakeDetection2", "i_Cyl-Home" := true, i_NextStationReady := "ST10_DBInterface_Stopper".Stopper[27].StationReady, i_PresentDelayTime := T#500ms, i_ReleaseDelayTime := T#500ms, io_NextyStopperStatus := "ST10_DBInterface_Stopper".Stopper[27].StopperStatus, io_Interface := "ST10_DBInterface_Stopper".Stopper[26], io_MotorCWRun :=, io_MotorCCWRun :=, o_StopperClyWP => "ST10Cylinder".Cy[48].Inout.AutoGoWork, o_StopperClyHP => "ST10Cylinder".Cy[48].Inout.AutoGoHome)
      I_Contact( "ST10_DBInterface_Stopper".Stopper[26].Done )
      Coil( "ST10_DBInterface_Stopper".Stopper[26].StopperRelease )
   END_RUNG
   // the same network as SCL:
   #Stopper[26](i_SysRun := "Station_Sys".Status.Run,   // "StopperCtrl"
                i_AutoMode := "Station_Sys".Auto.Mode,
                i_AutoRunnig := "Station_Sys".Auto.Running,
                i_Reset := "Station_Sys".Cmd.Reset,
                i_LineRunning := true,
                i_PalletArrivedNextStation := "iK-reserveTakeDetection3",
                i_StopperSensor := "iK-reserveTakeDetection2",
                "i_Cyl-Home" := true,
                i_NextStationReady := "ST10_DBInterface_Stopper".Stopper[27].StationReady,
                i_PresentDelayTime := T#500ms,
                i_ReleaseDelayTime := T#500ms,
                io_NextyStopperStatus := "ST10_DBInterface_Stopper".Stopper[27].StopperStatus,
                io_Interface := "ST10_DBInterface_Stopper".Stopper[26],
                o_StopperClyWP => "ST10Cylinder".Cy[48].Inout.AutoGoWork,
                o_StopperClyHP => "ST10Cylinder".Cy[48].Inout.AutoGoHome,
                ENO => #_w1);
   "ST10_DBInterface_Stopper".Stopper[26].StopperRelease := #_w1 AND NOT "ST10_DBInterface_Stopper".Stopper[26].Done;
END_REGION

REGION Network 26: H-shaftTakeStopperCylinder3 / K-reserveTakeStopperCylinder3
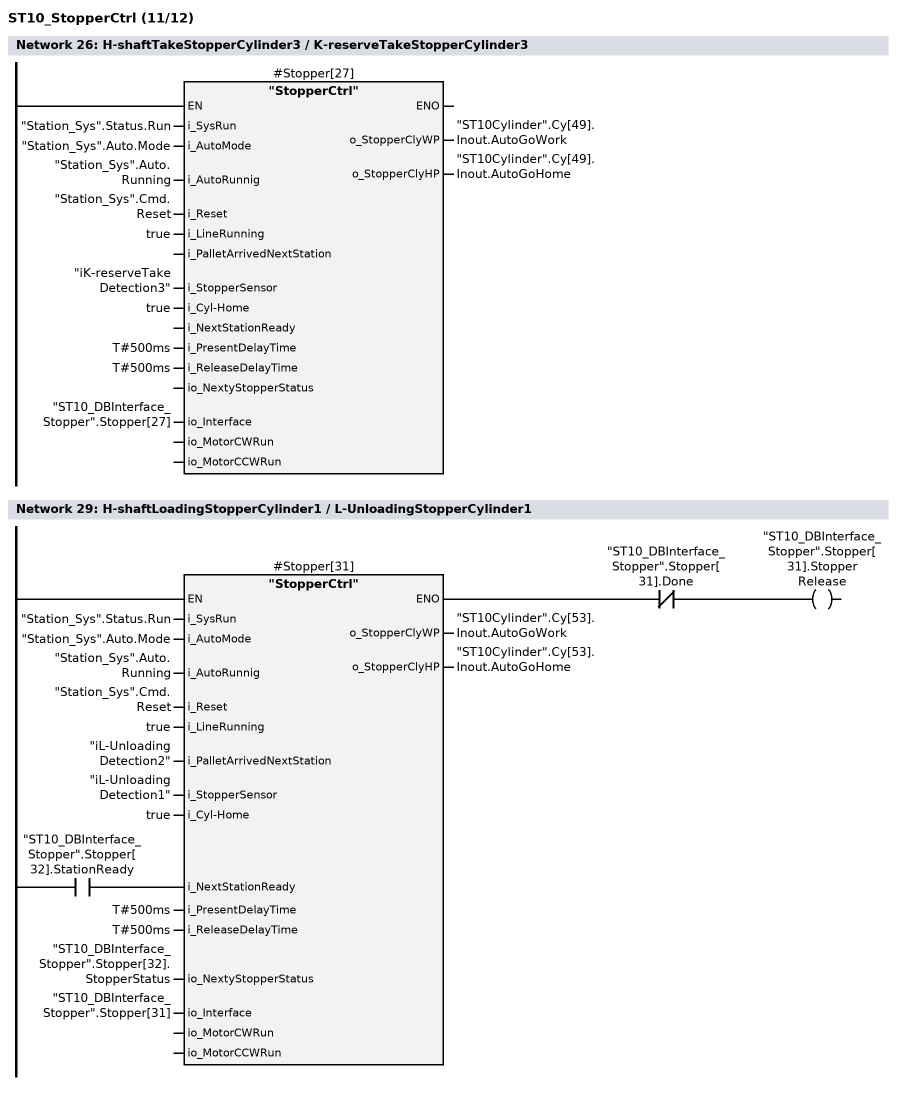
   RUNG wire#powerrail
      #Stopper[27](i_SysRun := "Station_Sys".Status.Run, i_AutoMode := "Station_Sys".Auto.Mode, i_AutoRunnig := "Station_Sys".Auto.Running, i_Reset := "Station_Sys".Cmd.Reset, i_LineRunning := true, i_PalletArrivedNextStation :=, i_StopperSensor := "iK-reserveTakeDetection3", "i_Cyl-Home" := true, i_NextStationReady :=, i_PresentDelayTime := T#500ms, i_ReleaseDelayTime := T#500ms, io_NextyStopperStatus :=, io_Interface := "ST10_DBInterface_Stopper".Stopper[27], io_MotorCWRun :=, io_MotorCCWRun :=, o_StopperClyWP => "ST10Cylinder".Cy[49].Inout.AutoGoWork, o_StopperClyHP => "ST10Cylinder".Cy[49].Inout.AutoGoHome)
   END_RUNG
   // the same network as SCL:
   #Stopper[27](i_SysRun := "Station_Sys".Status.Run,   // "StopperCtrl"
                i_AutoMode := "Station_Sys".Auto.Mode,
                i_AutoRunnig := "Station_Sys".Auto.Running,
                i_Reset := "Station_Sys".Cmd.Reset,
                i_LineRunning := true,
                i_StopperSensor := "iK-reserveTakeDetection3",
                "i_Cyl-Home" := true,
                i_PresentDelayTime := T#500ms,
                i_ReleaseDelayTime := T#500ms,
                io_Interface := "ST10_DBInterface_Stopper".Stopper[27],
                o_StopperClyWP => "ST10Cylinder".Cy[49].Inout.AutoGoWork,
                o_StopperClyHP => "ST10Cylinder".Cy[49].Inout.AutoGoHome);
END_REGION

REGION Network 27: -------------------------------------------------------------------------------------------------------------------------------
END_REGION

REGION Network 28: ------------------------------------------------------------------------------------------------------------------------------ / ------------------------------------------------ L -------------------------------------------------------------------------
END_REGION

REGION Network 29: H-shaftLoadingStopperCylinder1 / L-UnloadingStopperCylinder1
   RUNG wire#powerrail
      #Stopper[31](i_NextStationReady := wire#w1, i_SysRun := "Station_Sys".Status.Run, i_AutoMode := "Station_Sys".Auto.Mode, i_AutoRunnig := "Station_Sys".Auto.Running, i_Reset := "Station_Sys".Cmd.Reset, i_LineRunning := true, i_PalletArrivedNextStation := "iL-UnloadingDetection2", i_StopperSensor := "iL-UnloadingDetection1", "i_Cyl-Home" := true, i_PresentDelayTime := T#500ms, i_ReleaseDelayTime := T#500ms, io_NextyStopperStatus := "ST10_DBInterface_Stopper".Stopper[32].StopperStatus, io_Interface := "ST10_DBInterface_Stopper".Stopper[31], io_MotorCWRun :=, io_MotorCCWRun :=, o_StopperClyWP => "ST10Cylinder".Cy[53].Inout.AutoGoWork, o_StopperClyHP => "ST10Cylinder".Cy[53].Inout.AutoGoHome)
      I_Contact( "ST10_DBInterface_Stopper".Stopper[31].Done )
      Coil( "ST10_DBInterface_Stopper".Stopper[31].StopperRelease )
   END_RUNG
   RUNG wire#powerrail
      Contact( "ST10_DBInterface_Stopper".Stopper[32].StationReady )
   END_RUNG wire#w1
   // the same network as SCL:
   #Stopper[31](i_SysRun := "Station_Sys".Status.Run,   // "StopperCtrl"
                i_AutoMode := "Station_Sys".Auto.Mode,
                i_AutoRunnig := "Station_Sys".Auto.Running,
                i_Reset := "Station_Sys".Cmd.Reset,
                i_LineRunning := true,
                i_PalletArrivedNextStation := "iL-UnloadingDetection2",
                i_StopperSensor := "iL-UnloadingDetection1",
                "i_Cyl-Home" := true,
                i_NextStationReady := "ST10_DBInterface_Stopper".Stopper[32].StationReady,
                i_PresentDelayTime := T#500ms,
                i_ReleaseDelayTime := T#500ms,
                io_NextyStopperStatus := "ST10_DBInterface_Stopper".Stopper[32].StopperStatus,
                io_Interface := "ST10_DBInterface_Stopper".Stopper[31],
                o_StopperClyWP => "ST10Cylinder".Cy[53].Inout.AutoGoWork,
                o_StopperClyHP => "ST10Cylinder".Cy[53].Inout.AutoGoHome,
                ENO => #_w1);
   "ST10_DBInterface_Stopper".Stopper[31].StopperRelease := #_w1 AND NOT "ST10_DBInterface_Stopper".Stopper[31].Done;
END_REGION

REGION Network 30: H-shaftLoadingStopperCylinder2 / L-UnloadingStopperCylinder2
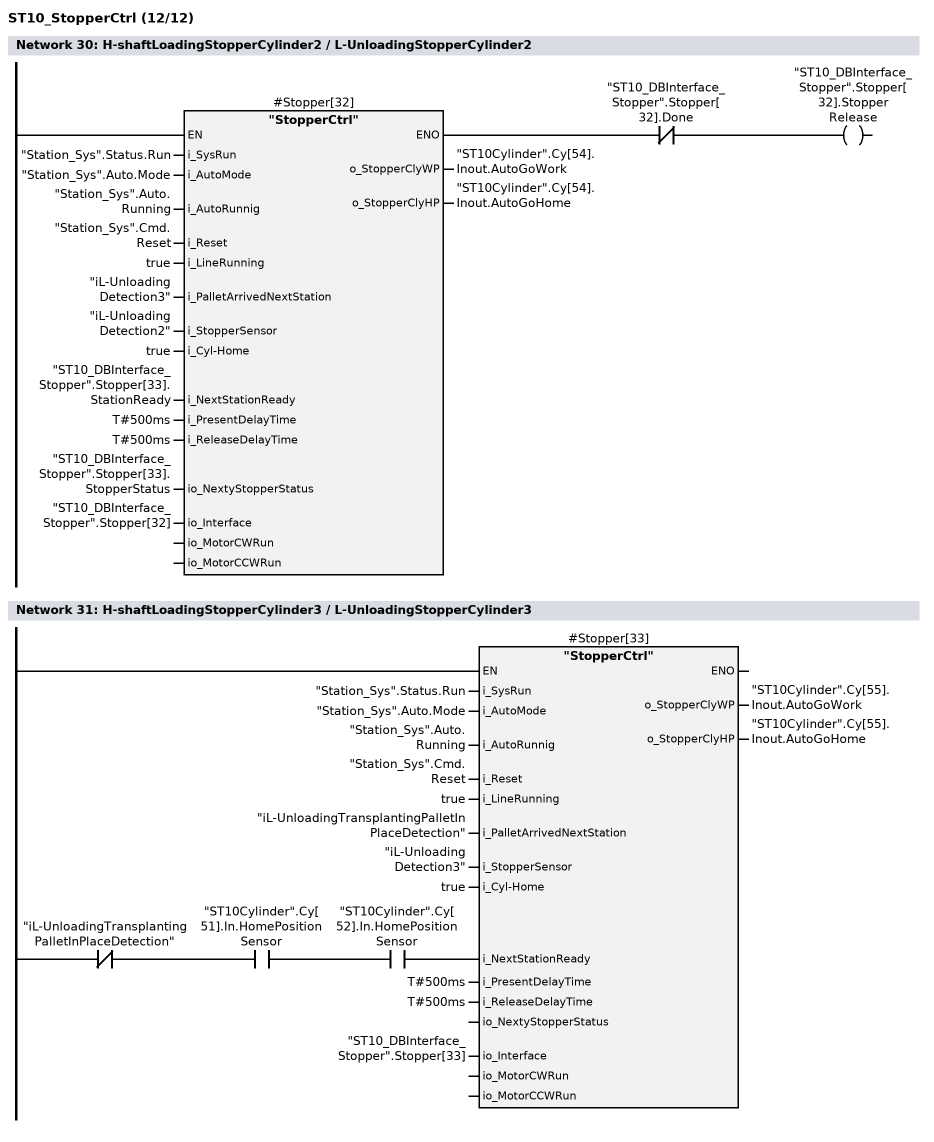
   RUNG wire#powerrail
      #Stopper[32](i_SysRun := "Station_Sys".Status.Run, i_AutoMode := "Station_Sys".Auto.Mode, i_AutoRunnig := "Station_Sys".Auto.Running, i_Reset := "Station_Sys".Cmd.Reset, i_LineRunning := true, i_PalletArrivedNextStation := "iL-UnloadingDetection3", i_StopperSensor := "iL-UnloadingDetection2", "i_Cyl-Home" := true, i_NextStationReady := "ST10_DBInterface_Stopper".Stopper[33].StationReady, i_PresentDelayTime := T#500ms, i_ReleaseDelayTime := T#500ms, io_NextyStopperStatus := "ST10_DBInterface_Stopper".Stopper[33].StopperStatus, io_Interface := "ST10_DBInterface_Stopper".Stopper[32], io_MotorCWRun :=, io_MotorCCWRun :=, o_StopperClyWP => "ST10Cylinder".Cy[54].Inout.AutoGoWork, o_StopperClyHP => "ST10Cylinder".Cy[54].Inout.AutoGoHome)
      I_Contact( "ST10_DBInterface_Stopper".Stopper[32].Done )
      Coil( "ST10_DBInterface_Stopper".Stopper[32].StopperRelease )
   END_RUNG
   // the same network as SCL:
   #Stopper[32](i_SysRun := "Station_Sys".Status.Run,   // "StopperCtrl"
                i_AutoMode := "Station_Sys".Auto.Mode,
                i_AutoRunnig := "Station_Sys".Auto.Running,
                i_Reset := "Station_Sys".Cmd.Reset,
                i_LineRunning := true,
                i_PalletArrivedNextStation := "iL-UnloadingDetection3",
                i_StopperSensor := "iL-UnloadingDetection2",
                "i_Cyl-Home" := true,
                i_NextStationReady := "ST10_DBInterface_Stopper".Stopper[33].StationReady,
                i_PresentDelayTime := T#500ms,
                i_ReleaseDelayTime := T#500ms,
                io_NextyStopperStatus := "ST10_DBInterface_Stopper".Stopper[33].StopperStatus,
                io_Interface := "ST10_DBInterface_Stopper".Stopper[32],
                o_StopperClyWP => "ST10Cylinder".Cy[54].Inout.AutoGoWork,
                o_StopperClyHP => "ST10Cylinder".Cy[54].Inout.AutoGoHome,
                ENO => #_w1);
   "ST10_DBInterface_Stopper".Stopper[32].StopperRelease := #_w1 AND NOT "ST10_DBInterface_Stopper".Stopper[32].Done;
END_REGION

REGION Network 31: H-shaftLoadingStopperCylinder3 / L-UnloadingStopperCylinder3
   RUNG wire#powerrail
      #Stopper[33](i_NextStationReady := wire#w1, i_SysRun := "Station_Sys".Status.Run, i_AutoMode := "Station_Sys".Auto.Mode, i_AutoRunnig := "Station_Sys".Auto.Running, i_Reset := "Station_Sys".Cmd.Reset, i_LineRunning := true, i_PalletArrivedNextStation := "iL-UnloadingTransplantingPalletInPlaceDetection", i_StopperSensor := "iL-UnloadingDetection3", "i_Cyl-Home" := true, i_PresentDelayTime := T#500ms, i_ReleaseDelayTime := T#500ms, io_NextyStopperStatus :=, io_Interface := "ST10_DBInterface_Stopper".Stopper[33], io_MotorCWRun :=, io_MotorCCWRun :=, o_StopperClyWP => "ST10Cylinder".Cy[55].Inout.AutoGoWork, o_StopperClyHP => "ST10Cylinder".Cy[55].Inout.AutoGoHome)
   END_RUNG
   RUNG wire#powerrail
      I_Contact( "iL-UnloadingTransplantingPalletInPlaceDetection" )
      Contact( "ST10Cylinder".Cy[51].In.HomePositionSensor )
      Contact( "ST10Cylinder".Cy[52].In.HomePositionSensor )
   END_RUNG wire#w1
   // the same network as SCL:
   #Stopper[33](i_SysRun := "Station_Sys".Status.Run,   // "StopperCtrl"
                i_AutoMode := "Station_Sys".Auto.Mode,
                i_AutoRunnig := "Station_Sys".Auto.Running,
                i_Reset := "Station_Sys".Cmd.Reset,
                i_LineRunning := true,
                i_PalletArrivedNextStation := "iL-UnloadingTransplantingPalletInPlaceDetection",
                i_StopperSensor := "iL-UnloadingDetection3",
                "i_Cyl-Home" := true,
                i_NextStationReady := NOT "iL-UnloadingTransplantingPalletInPlaceDetection" AND "ST10Cylinder".Cy[51].In.HomePositionSensor AND "ST10Cylinder".Cy[52].In.HomePositionSensor,
                i_PresentDelayTime := T#500ms,
                i_ReleaseDelayTime := T#500ms,
                io_Interface := "ST10_DBInterface_Stopper".Stopper[33],
                o_StopperClyWP => "ST10Cylinder".Cy[55].Inout.AutoGoWork,
                o_StopperClyHP => "ST10Cylinder".Cy[55].Inout.AutoGoHome);
END_REGION

REGION Network 32: -------------------------------------------------------------------------------------------------------------------------------
END_REGION
END_FUNCTION_BLOCK
